Universal Robots PolyScope program: program.urp

Program program (installation=default directory=/ursim/programs createdIn=5.15.2 lastSavedIn=5.15.2 robotSerialNumber=20195599999)
Calibrated DH parameters: a=[0, -0.425, -0.3922, 0, 0, 0]; d=[0.1625, 0, 0, 0.1333, 0.0997, 0.0996]; alpha=[1.570796, 0, 0, 1.570796, -1.570796, 0]; deltaTheta=[0, 0, 0, 0, 0, 0]
InitVariablesNode
Robot Program (runOnlyOnce=false)
  Script file /ursim/programs/script_code.script
    |             a=[0,0,0,0,0,0]
    |             movej(a)
    |             b=[1,0,0,0,0,0]
    |             movej(b)
    |             c=[0,-1,0,0,0,0]
    |             movej(c)
  Halt
